# EPICS substitutions: gigeApp/Db/pluginROI.substitutions
#
# pluginROI.substitutions
#

file NDPluginBase.template
{
	{
	P=$(CAM):,
	R=ROI$(N):,
	PORT=$(CAM_PORT).ROI$(N),
	ADDR=0,
	TIMEOUT=1,
	NDARRAY_PORT=$(PLUGIN_SRC),
	NDARRAY_ADDR=0
	}
}

file NDROI.template
{
	{
	P=$(CAM):,
	R=ROI$(N):,
	PORT=$(CAM_PORT).ROI$(N),
	ADDR=0,
	TIMEOUT=1
	}
}
